Fanuc KAREL source: WRITE_DICT.kl

PROGRAM T
%NOLOCKGROUP
VAR
 v0 : FILE
 v1 : STRING[40]
 v2 : INTEGER
 v3 : INTEGER
BEGIN
 WRITE_DICT(v0, v1, v2, v3)
END T
